DATA_BLOCK "DB_ActiveConfigModel"
{ S7_Optimized_Access := 'TRUE' }
VERSION : 0.1
NON_RETAIN
   VAR
      Data : "UDT_ActiveConfigModel";
   END_VAR

BEGIN
END_DATA_BLOCK
